ABB RobotStudio station: RobotSimulator_PixelProject.rspag

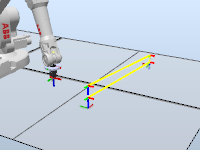
--- station ---
Station Final_project (saved by RobotStudio 7.0.8666.559)
Controller IRB_1600_6kg_1.45m
  mechanical unit ROB_1: IRB1600_6_145__02, 6 joints, base frame (0, 0, 0) mm
Layout (positions relative to the parent item):
  - IRB1600_6_145__02 [mechanism, from Robots\IRB1600_6_145_G_02.rslib] at (0, 0, 0) mm; joint values [-1.991, 0.9649, 0.1667, 0, 0.4392, -3.5618] (rad or m)
  - GS25_ParallelGripper [mechanism, from Libraries\GS25_ParallelGripper.rslib] at (-400, -895.2, 277.08) mm, rotated rx 180 ry 0 rz -90 deg
Attachment: GS25_ParallelGripper is attached to IRB1600_6_145__02 / Link6
Targets, tools, work objects and paths stored in the station and not in the controller backup, written as RAPID:
! task T_ROB1
MODULE Module1
  CONST jointtarget Home:=[[0,0,0,0,45,0],[9E+09,9E+09,9E+09,9E+09,9E+09,9E+09]];
ENDMODULE


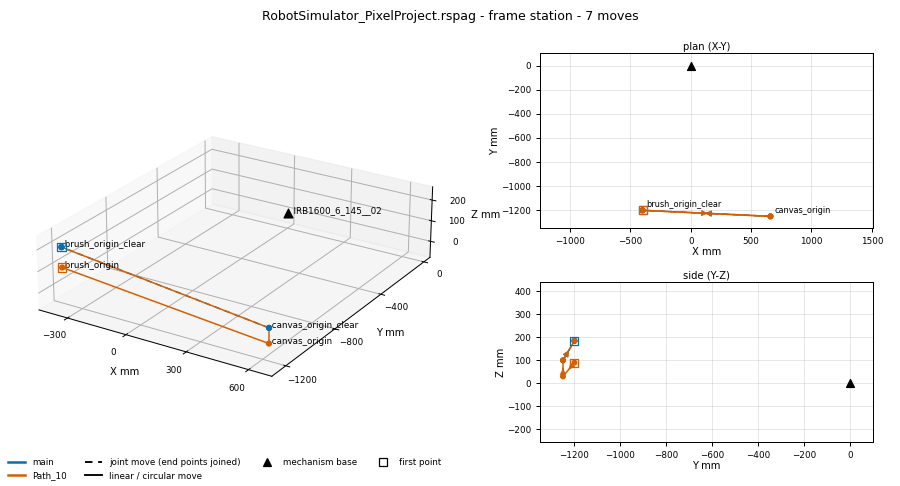
[picture p0: tool path of RobotSimulator_PixelProject.rspag in frame station, 7 of 19 moves have a stored position in this frame; points joined in program order, loops and branches not executed]
--- Backups/IRB_1600_6kg_1.45m/RAPID/TASK1/PROGMOD/CalibData.mod ---
MODULE CalibData
	PERS tooldata GS25_ParallelGripper:=[TRUE,[[0,0,92.075],[1,0,0,0]],[1,[0,0,45],[1,0,0,0],0,0,0]];
	PERS wobjdata wobj_brush:=[FALSE,TRUE,"",[[-400,-1200,0],[1,0,0,0]],[[0,0,0],[1,0,0,0]]];
	PERS wobjdata wobj_canvas:=[FALSE,TRUE,"",[[660,-1250,0],[0.707106781,0,0,0.707106781]],[[0,0,0],[1,0,0,0]]];
ENDMODULE

--- Backups/IRB_1600_6kg_1.45m/RAPID/TASK1/PROGMOD/Module1.mod ---
MODULE Module1
    CONST robtarget brush_origin:=[[0,0,90],[0,-0.707106781,0.707106781,0],[-2,0,-2,0],[9E+09,9E+09,9E+09,9E+09,9E+09,9E+09]];
    CONST robtarget canvas_origin:=[[0,0,30],[0,0,1,0],[-1,0,-1,0],[9E+09,9E+09,9E+09,9E+09,9E+09,9E+09]];
	CONST robtarget canvas_origin_clear:=[[0,0,100],[0,0,1,0],[-1,0,-1,0],[9E+09,9E+09,9E+09,9E+09,9E+09,9E+09]];
	CONST robtarget brush_origin_clear:=[[0,0,185],[0,-0.707106781,0.707106781,0],[-2,0,-2,0],[9E+09,9E+09,9E+09,9E+09,9E+09,9E+09]];
    !***********************************************************
    ! Module:  Module1
    ! Description:
    !   <Insert description here>
    ! Author: Thomas
    ! Version: 1.0
    !***********************************************************
    PROC Open_gripper()
        SetDO D652_10_DO1, 0;
        WaitTime 0.5;
    ENDPROC
    PROC Close_gripper()
        SetDO D652_10_DO1, 1;
        WaitTime 0.5;
    ENDPROC
    PROC main()
        !MoveJ brush_origin,v1000,z100,GS25_ParallelGripper\WObj:=wobj_brush;
        VAR string currentline;
        VAR bool looping;
        VAR iodev infile;
        VAR string xPosstr;
        VAR string yPosstr;
        VAR num xPos;
        VAR num yPos;
        VAR num found;
        VAR num strlength;
        VAR bool randomthing1;
        VAR bool randomthing2;
        VAR num brushNum := 0;
        VAR num brushSize:= 21;!21;!position is in inches, set to 25 before.
        VAR num pickupSize:= 50.8;
        Open "HOME:/finalfinalfinalrobotStudioVals.txt", infile\Read;
        looping:= TRUE;
        MoveJ brush_origin_clear,v1000,z100,GS25_ParallelGripper\WObj:=wobj_brush;
        MoveL RelTool (brush_origin_clear, 0, brushNum*brushSize, 0),v100,z100,GS25_ParallelGripper\WObj:=wobj_brush;
        MoveL RelTool (brush_origin, 0, brushNum*brushSize, 0),v100,fine,GS25_ParallelGripper\WObj:=wobj_brush;
        MoveL RelTool (brush_origin_clear, 0, brushNum*brushSize, 0),v100,z100,GS25_ParallelGripper\WObj:=wobj_brush;
        MoveL canvas_origin_clear,v1000,z100,GS25_ParallelGripper\WObj:=wobj_canvas;
        WHILE looping DO
            currentline := ReadStr(infile);
            IF currentline = EOF THEN
               TPWrite "The file is empty";
               looping := FALSE;
            ELSE
                TPWrite currentline;
                IF currentline = "end" THEN
                    brushNum := brushNum + 1;
                    MoveJ brush_origin_clear,v1000,z100,GS25_ParallelGripper\WObj:=wobj_brush;
                    MoveL RelTool (brush_origin_clear, -(brushNum-1)*pickupSize, 0, 0),v100,z100,GS25_ParallelGripper\WObj:=wobj_brush;
                    MoveL RelTool (brush_origin, -(brushNum-1)*pickupSize, 0, 0),v100,fine,GS25_ParallelGripper\WObj:=wobj_brush;
                    Open_gripper;
                    MoveL RelTool (brush_origin_clear, -(brushNum-1)*pickupSize, 0, 0),v100,z100,GS25_ParallelGripper\WObj:=wobj_brush;
                    MoveL RelTool (brush_origin_clear, -brushNum*pickupSize, 0, 0),v100,z100,GS25_ParallelGripper\WObj:=wobj_brush;
                    MoveL RelTool (brush_origin, -brushNum*pickupSize, 0, 0),v100,fine,GS25_ParallelGripper\WObj:=wobj_brush;
                    Close_gripper;
                    MoveL RelTool (brush_origin_clear, -brushNum*pickupSize, 0, 0),v100,z100,GS25_ParallelGripper\WObj:=wobj_brush;

                ELSE
                    found := StrFind(currentline,1,"  ");
                    strlength := StrLen(currentline);
                    xPosstr:= StrPart(currentline,1,found-1);
                    TPWrite xPosstr;
                    yPosstr:= StrPart(currentline,found+2,strlength+1-(found+2));
                    TPWrite yPosstr;
                    randomthing1 := StrToVal(xPosstr,xPos);
                    randomthing2 := StrToVal(yPosstr,yPos);
                    IF (NOT randomthing1) OR (NOT randomthing2) THEN
                        TPWrite "Error converting string to number";
                        looping := FALSE;
                    ENDIF
                    MoveJ RelTool (canvas_origin_clear, -xPos*brushSize, yPos*brushSize, 0),v100,z100,GS25_ParallelGripper\WObj:=wobj_canvas;
                    MoveL RelTool (canvas_origin, -xPos*brushSize, yPos*brushSize, 0),v100,fine,GS25_ParallelGripper\WObj:=wobj_canvas;
                    MoveL RelTool (canvas_origin_clear, -xPos*brushSize, yPos*brushSize, 0),v100,z100,GS25_ParallelGripper\WObj:=wobj_canvas;

                ENDIF
            ENDIF





        ENDWHILE


    ENDPROC
    PROC getBrush()

    ENDPROC

    PROC Stamp()

    ENDPROC

    PROC Path_10()
        MoveL brush_origin,v1000,z100,GS25_ParallelGripper\WObj:=wobj_brush;
        MoveL canvas_origin,v1000,z100,GS25_ParallelGripper\WObj:=wobj_canvas;
		MoveL canvas_origin_clear,v1000,z100,GS25_ParallelGripper\WObj:=wobj_canvas;
		MoveL brush_origin_clear,v1000,z100,GS25_ParallelGripper\WObj:=wobj_brush;
    ENDPROC

ENDMODULE

--- Backups/IRB_1600_6kg_1.45m/SYSPAR/EIO.cfg ---
EIO:CFG_1.0:6:1::
#
EIO_SIGNAL:

      -Name "D652_10_DO1" -SignalType "DO"
